PROGRAM P_Sample
VAR CONSTANT
	sNetID						: T_AmsNetId 	:= '5.125.236.17.2.1'; // EtherCAT Master AMS NetID
	sModule_GUID				: STRING(36)	:= '28111931-0002-0000-5230-FE1A00001500';
END_VAR
VAR
	fbSafeDiag_Diagnostic		: FB_SafeDiag_Diagnostic;
	stSafeDiag					: ST_EL6910_SafeDiag;
	bExecute					: BOOL			:= TRUE;
END_VAR

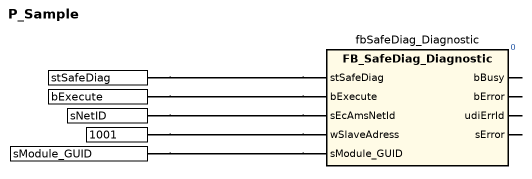
fbSafeDiag_Diagnostic(
    stSafeDiag := stSafeDiag,
    bExecute := bExecute,
    sEcAmsNetId := sNetID,
    wSlaveAdress := 1001,
    sModule_GUID := sModule_GUID); // FB_SafeDiag_Diagnostic

END_PROGRAM

(* stored: Version 1.1.0.1, ProductVersion 3.1.4024.12
   POU P_Sample: Id {40f4095b-58b8-4f55-820b-3c5d26950fec}, SpecialFunc None *)
